PROGRAM MAIN
VAR
END_VAR

END_PROGRAM

(* stored: Version 1.1.0.1
   POU MAIN: Id {f742d04b-4425-48cc-8bf5-cb3b9598befa} *)
